{attribute addProperty BoxType "EL5001-0000-1017"}
{attribute addProperty Id "SSI_InputsAT %I*SSI_Inputs_F7D238D14860WcStateAT %I*WcState_F855686C1620InfoDataAT %I*InfoData_BC63D37F80100"}
{attribute addProperty CRC "3547044431"}
{attribute addProperty SizeInBites "144"}
{attribute addProperty SizeInBytes "18"}
TYPE EL5001_5BDAD4AF :
STRUCT
	{attribute addProperty Name "SSI_Inputs"}
	SSI_Inputs : SSI_Inputs_F7D238D1;
	{attribute addProperty Name "WcState"}
	WcState : WcState_F855686C;
	{attribute addProperty Name "InfoData"}
	InfoData : InfoData_BC63D37F;
END_STRUCT
END_TYPE

(* stored: Version 1.2.0.0, ProductVersion 3.1.4024.9
   DUT EL5001_5BDAD4AF: Id {ce34307e-dfa0-4c37-88ff-5766bacd20bb} *)
